Universal Robots PolyScope program: CommPlotNoWaits.urp

Program CommPlotNoWaits (installation=botross directory=/programs/APS2OsUltimosRomanticos createdIn=3.15.3.106223 lastSavedIn=3.15.3.106223 robotSerialNumber=2017357017)
Calibrated DH parameters: a=[0.0001, -0.032836, -0.39033, 0.000086, 0.000053, 0]; d=[0.089393, 264.548863, -261.578988, -2.85966, 0.094927, 0.082356]; alpha=[1.569373, -0.001603, 0.013671, 1.570599, -1.570158, 0]; deltaTheta=[0.000031, -1.49356, 1.597104, -0.103695, -0.000023, -0.000043]
BeforeStart
  Socket := socket_open("10.103.16.140",20000)
  Num_points := socket_read_ascii_float(1)
Robot Program (runOnlyOnce=false)
  Loop While (checkContinuously=false) expression=Socket≟ False
    Socket := socket_open("10.103.16.140",20000)
  Num_points := socket_read_ascii_float(1)
  N := Num_points[1]
  X := socket_read_ascii_float(N)
  Y := socket_read_ascii_float(N)
  Z := socket_read_ascii_float(N)
  count := 1
  Loop While (checkContinuously=false) expression=count<N
    move2pose := p[X[count]/5000,Y[count]/5000,Z[count]/1000,0,0,0]
    MoveL speed 250 mm/s, acceleration 1200 mm/s^2 (useActiveTCP=true) feature=Plano_BotRoss
      Waypoint Waypoint (Variable): variable=move2pose
    count := count+1
